PROGRAM EXAMPLES_PRG
VAR
	_context : fbContext;
END_VAR

_context.Run();

END_PROGRAM

(* stored: Version 1.1.0.1, ProductVersion 3.1.4024.6
   POU EXAMPLES_PRG: Id {74d7366d-b6fb-47e3-acf3-d19ebdfb665f}, SpecialFunc None *)
